TYPE S_POSITION3D EXTENDS S_POSITION2D :
STRUCT
	Z : LREAL;
END_STRUCT
END_TYPE

(* stored: Version 1.1.0.1, ProductVersion 3.1.4019.2
   DUT S_POSITION3D: Id {f7e81338-0cae-4d93-aefb-7684ca59a3a1} *)
